PROGRAM MAIN
VAR
	rWriteAnalog1 : REAL;
	rWriteAnalog2 : REAL;
END_VAR

GVL.bAnalog_Outputs[1] := REAL_TO_INT(rWriteAnalog1/10*32767);
GVL.bAnalog_Outputs[2] := REAL_TO_INT(rWriteAnalog2/10*32767);

END_PROGRAM

(* stored: Version 1.1.0.1, ProductVersion 3.1.4024.12
   POU MAIN: Id {dba29591-cf21-4385-93d4-070326345606}, SpecialFunc None *)
